Yaskawa INFORM job: small_pipe_cylinder_program.JBI

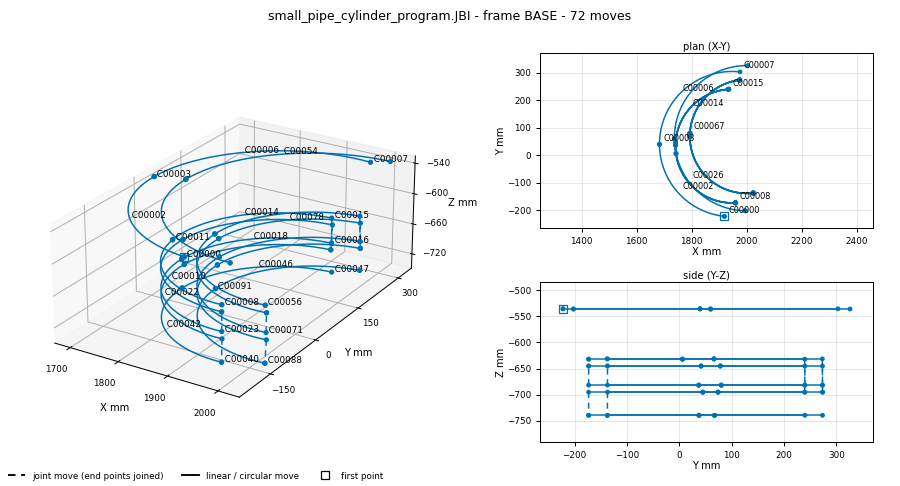
[picture p0: tool path of small_pipe_cylinder_program.JBI in frame BASE, 72 of 105 moves have a stored position in this frame; points joined in program order, loops and branches not executed]
/JOB
//NAME small_pipe_cylinder_program
//POS
///NPOS 96,0,96,0,0,0
///TOOL 0
///POSTYPE BASE
///RECTAN
///RCONF 0,0,0,0,0,0,0,0,0,0,0,0,0,0,0,0,0,0,0,0,0,0,0,0
C00000=1919.180043,-222.253565,-535.692960,175.000000,-60.000000,83.854678
C00001=1919.180043,-222.253565,-535.692960,175.000000,-60.000000,83.854678
C00002=1752.178281,-137.536841,-535.692960,175.000000,-60.000000,42.349745
C00003=1683.223907,39.648654,-535.692960,175.000000,-60.000000,5.000000
C00004=1683.223907,39.648654,-535.692960,175.000000,-60.000000,5.000000
C00005=1683.223907,39.648654,-535.692960,175.000000,-60.000000,5.000000
C00006=1753.745394,220.186963,-535.692960,-175.000000,-60.000000,-42.851744
C00007=1976.266389,303.143966,-535.692960,175.000000,-60.000000,-96.256814
C00008=1960.191811,-173.203258,-631.848500,-86.734427,-89.999999,5.000000
C00009=1960.191811,-173.203258,-631.848500,-86.734427,-89.999999,5.000000
C00010=1829.996385,-136.308422,-631.848500,-124.908956,-89.999999,5.000000
C00011=1743.293664,6.153364,-631.848500,-172.441376,-89.999999,5.000000
C00012=1743.293664,6.153364,-631.848500,-172.441376,-89.999999,5.000000
C00013=1743.293664,6.153364,-631.848500,-172.441376,-89.999999,5.000000
C00014=1789.234673,165.568202,-631.848500,140.288971,-90.000000,5.000000
C00015=1933.789573,239.763101,-631.848500,94.050669,-90.000000,5.000000
C00016=1934.344025,239.801617,-681.511500,93.896764,-90.000000,5.000000
C00017=1934.344025,239.801617,-681.511500,93.896764,-90.000000,5.000000
C00018=1800.374217,177.933006,-681.511500,135.679176,-89.999999,5.000000
C00019=1741.530247,37.146701,-681.511500,175.000000,-89.999999,5.000000
C00020=1741.530247,37.146701,-681.511500,175.000000,-89.999999,5.000000
C00021=1741.530247,37.146701,-681.511500,175.000000,-89.999999,5.000000
C00022=1796.795260,-107.434295,-681.511500,-137.116260,-90.000000,5.000000
C00023=1960.117862,-173.207464,-681.511500,-86.754938,-89.999999,5.000000
C00024=1959.976972,-173.215404,-645.009960,-175.000000,-60.000000,93.205986
C00025=1959.976972,-173.215404,-645.009960,-175.000000,-60.000000,93.205986
C00026=1788.368845,-97.777979,-645.009960,175.000000,-60.000000,39.334277
C00027=1741.661984,41.661903,-645.009960,175.000000,-60.000000,-5.000000
C00028=1741.661984,41.661903,-645.009960,175.000000,-60.000000,-5.000000
C00029=1741.661984,41.661903,-645.009960,175.000000,-60.000000,-5.000000
C00030=1803.493991,181.060147,-645.009960,-175.000000,-60.000000,-45.544034
C00031=1935.364811,239.868614,-645.009960,175.000000,-60.000000,-86.386512
C00032=1933.055266,239.709788,-694.950460,-175.000000,-60.000000,-85.745457
C00033=1933.055266,239.709788,-694.950460,-175.000000,-60.000000,-85.745457
C00034=1804.782266,182.313251,-694.950460,175.000000,-60.000000,-46.041702
C00035=1741.813609,44.834284,-694.950460,175.000000,-60.000000,-5.000000
C00036=1741.813609,44.834284,-694.950460,175.000000,-60.000000,-5.000000
C00037=1741.813609,44.834284,-694.950460,175.000000,-60.000000,-5.000000
C00038=1793.336318,-103.615645,-694.950460,175.000000,-60.000000,41.456964
C00039=1960.430374,-173.189508,-694.950460,175.000000,-60.000000,93.331743
C00040=1959.364741,-173.248787,-739.065960,-175.000000,-60.000000,93.036200
C00041=1959.364741,-173.248787,-739.065960,-175.000000,-60.000000,93.036200
C00042=1802.374489,-113.212580,-739.065960,-175.000000,-60.000000,45.108096
C00043=1741.538277,37.563554,-739.065960,175.000000,-60.000000,-5.000000
C00044=1741.538277,37.563554,-739.065960,175.000000,-60.000000,-5.000000
C00045=1741.538277,37.563554,-739.065960,175.000000,-60.000000,-5.000000
C00046=1807.515538,184.901335,-739.065960,-175.000000,-60.000000,-47.084060
C00047=1935.638086,239.885690,-739.065960,175.000000,-60.000000,-86.462333
C00048=1995.134330,-202.194927,-536.078460,175.000000,-60.000000,88.606450
C00049=1995.134330,-202.194927,-536.078460,175.000000,-60.000000,88.606450
C00050=1813.082954,-123.234912,-536.078460,175.000000,-60.000000,44.498499
C00051=1737.325476,59.695630,-536.078460,-175.000000,-60.000000,5.000000
C00052=1737.325476,59.695630,-536.078460,-175.000000,-60.000000,5.000000
C00053=1737.325476,59.695630,-536.078460,-175.000000,-60.000000,5.000000
C00054=1817.601589,251.667664,-536.078460,-175.000000,-60.000000,-45.879584
C00055=2004.328239,326.202425,-536.078460,-175.000000,-60.000000,-90.600098
C00056=2023.008270,-137.447122,-631.340500,-83.760239,-90.000000,5.000000
C00057=2023.008270,-137.447122,-631.340500,-83.760239,-90.000000,5.000000
C00058=1844.451298,-67.609986,-631.340500,-138.962647,-89.999999,5.000000
C00059=1793.619781,66.206992,-631.340500,-175.000000,-89.999999,5.000000
C00060=1793.619781,66.206992,-631.340500,-175.000000,-89.999999,5.000000
C00061=1793.619781,66.206992,-631.340500,-175.000000,-89.999999,5.000000
C00062=1827.332269,181.452385,-631.340500,146.826604,-89.999999,5.000000
C00063=1973.123011,273.324532,-631.340500,97.608744,-89.999999,5.000000
C00064=1974.788266,273.540110,-681.475500,97.143765,-90.000000,5.000000
C00065=1974.788266,273.540110,-681.475500,97.143765,-90.000000,5.000000
C00066=1849.340238,209.503950,-681.475500,136.941193,-90.000000,5.000000
C00067=1793.957901,80.233327,-681.475500,175.000000,-90.000000,5.000000
C00068=1793.957901,80.233327,-681.475500,175.000000,-90.000000,5.000000
C00069=1793.957901,80.233327,-681.475500,175.000000,-90.000000,5.000000
C00070=1870.223695,-92.494769,-681.475500,-129.029688,-90.000000,5.000000
C00071=2024.730486,-137.251517,-681.475500,-83.280269,-90.000000,5.000000
C00072=2025.322950,-137.180845,-644.921960,175.000000,-60.000000,96.884954
C00073=2025.322950,-137.180845,-644.921960,175.000000,-60.000000,96.884954
C00074=1848.138782,-71.733732,-644.921960,175.000000,-60.000000,42.569271
C00075=1793.863419,78.477670,-644.921960,-175.000000,-60.000000,-5.000000
C00076=1793.863419,78.477670,-644.921960,-175.000000,-60.000000,-5.000000
C00077=1793.863419,78.477670,-644.921960,-175.000000,-60.000000,-5.000000
C00078=1854.789412,215.118781,-644.921960,-175.000000,-60.000000,-45.225583
C00079=1974.546352,273.509645,-644.921960,-175.000000,-60.000000,-82.788717
C00080=1975.515287,273.629922,-694.925960,-175.000000,-60.000000,-83.059086
C00081=1975.515287,273.629922,-694.925960,-175.000000,-60.000000,-83.059086
C00082=1852.242914,212.547679,-694.925960,175.000000,-60.000000,-44.223499
C00083=1793.692664,74.091023,-694.925960,175.000000,-60.000000,-5.000000
C00084=1793.692664,74.091023,-694.925960,175.000000,-60.000000,-5.000000
C00085=1793.692664,74.091023,-694.925960,175.000000,-60.000000,-5.000000
C00086=1859.683120,-83.344030,-694.925960,175.000000,-60.000000,47.104301
C00087=2025.338332,-137.178987,-694.925960,-175.000000,-60.000000,96.889245
C00088=2022.883642,-137.460710,-739.166460,175.000000,-60.000000,96.205045
C00089=2022.883642,-137.460710,-739.166460,175.000000,-60.000000,96.205045
C00090=1857.753393,-81.527923,-739.166460,175.000000,-60.000000,46.370500
C00091=1793.612010,67.285889,-739.166460,175.000000,-60.000000,5.000000
C00092=1793.612010,67.285889,-739.166460,175.000000,-60.000000,5.000000
C00093=1793.612010,67.285889,-739.166460,175.000000,-60.000000,5.000000
C00094=1851.248443,211.518786,-739.166460,175.000000,-60.000000,-43.827253
C00095=1975.230312,273.595029,-739.166460,175.000000,-60.000000,-82.979584
///POSTYPE PULSE
///PULSE
EX00000=86016.0
EX00001=95232.0
EX00002=275456.0
EX00003=283648.0
///POSTYPE PULSE
///PULSE
EC00000=86016.0
EC00001=86016.0
EC00002=86016.0
EC00003=86016.0
EC00004=86016.0
EC00005=86016.0
EC00006=86016.0
EC00007=86016.0
EC00008=95232.0
EC00009=95232.0
EC00010=95232.0
EC00011=95232.0
EC00012=95232.0
EC00013=95232.0
EC00014=95232.0
EC00015=95232.0
EC00016=95232.0
EC00017=95232.0
EC00018=95232.0
EC00019=95232.0
EC00020=95232.0
EC00021=95232.0
EC00022=95232.0
EC00023=95232.0
EC00024=95232.0
EC00025=95232.0
EC00026=95232.0
EC00027=95232.0
EC00028=95232.0
EC00029=95232.0
EC00030=95232.0
EC00031=95232.0
EC00032=95232.0
EC00033=95232.0
EC00034=95232.0
EC00035=95232.0
EC00036=95232.0
EC00037=95232.0
EC00038=95232.0
EC00039=95232.0
EC00040=95232.0
EC00041=95232.0
EC00042=95232.0
EC00043=95232.0
EC00044=95232.0
EC00045=95232.0
EC00046=95232.0
EC00047=95232.0
EC00048=275456.0
EC00049=275456.0
EC00050=275456.0
EC00051=275456.0
EC00052=275456.0
EC00053=275456.0
EC00054=275456.0
EC00055=275456.0
EC00056=283648.0
EC00057=283648.0
EC00058=283648.0
EC00059=283648.0
EC00060=283648.0
EC00061=283648.0
EC00062=283648.0
EC00063=283648.0
EC00064=283648.0
EC00065=283648.0
EC00066=283648.0
EC00067=283648.0
EC00068=283648.0
EC00069=283648.0
EC00070=283648.0
EC00071=283648.0
EC00072=283648.0
EC00073=283648.0
EC00074=283648.0
EC00075=283648.0
EC00076=283648.0
EC00077=283648.0
EC00078=283648.0
EC00079=283648.0
EC00080=283648.0
EC00081=283648.0
EC00082=283648.0
EC00083=283648.0
EC00084=283648.0
EC00085=283648.0
EC00086=283648.0
EC00087=283648.0
EC00088=283648.0
EC00089=283648.0
EC00090=283648.0
EC00091=283648.0
EC00092=283648.0
EC00093=283648.0
EC00094=283648.0
EC00095=283648.0
//INST
///DATE 2023/08/16 14:27
///ATTR SC,RW,RJ
////FRAME BASE
///GROUP1 RB1,ST1
NOP
MOVJ P009 EX000 VJ=15.00
MOVJ C00000 EC00000 VJ=15.0
CALL JOB:SPYON
MOVC C00001 EC00001 V=150.0
MOVC C00002 EC00002 V=150.0
MOVC C00003 EC00003 V=150.0
MOVJ C00004 EC00004 VJ=15.0
MOVC C00005 EC00005 V=150.0
MOVC C00006 EC00006 V=150.0
MOVC C00007 EC00007 V=150.0
CALL JOB:SPYOF
MOVJ P009 VJ=15.00
MOVL P009 EX00000 V=150.0
MOVJ C00008 EC00008 VJ=15.0
CALL JOB:SPYON
MOVC C00009 EC00009 V=150.0
MOVC C00010 EC00010 V=150.0
MOVC C00011 EC00011 V=150.0
MOVJ C00012 EC00012 VJ=15.0
MOVC C00013 EC00013 V=150.0
MOVC C00014 EC00014 V=150.0
MOVC C00015 EC00015 V=150.0
MOVJ C00016 EC00016 VJ=15.0
MOVC C00017 EC00017 V=150.0
MOVC C00018 EC00018 V=150.0
MOVC C00019 EC00019 V=150.0
MOVJ C00020 EC00020 VJ=15.0
MOVC C00021 EC00021 V=150.0
MOVC C00022 EC00022 V=150.0
MOVC C00023 EC00023 V=150.0
MOVJ C00024 EC00024 VJ=15.0
MOVC C00025 EC00025 V=150.0
MOVC C00026 EC00026 V=150.0
MOVC C00027 EC00027 V=150.0
MOVJ C00028 EC00028 VJ=15.0
MOVC C00029 EC00029 V=150.0
MOVC C00030 EC00030 V=150.0
MOVC C00031 EC00031 V=150.0
MOVJ C00032 EC00032 VJ=15.0
MOVC C00033 EC00033 V=150.0
MOVC C00034 EC00034 V=150.0
MOVC C00035 EC00035 V=150.0
MOVJ C00036 EC00036 VJ=15.0
MOVC C00037 EC00037 V=150.0
MOVC C00038 EC00038 V=150.0
MOVC C00039 EC00039 V=150.0
MOVJ C00040 EC00040 VJ=15.0
MOVC C00041 EC00041 V=150.0
MOVC C00042 EC00042 V=150.0
MOVC C00043 EC00043 V=150.0
MOVJ C00044 EC00044 VJ=15.0
MOVC C00045 EC00045 V=150.0
MOVC C00046 EC00046 V=150.0
MOVC C00047 EC00047 V=150.0
CALL JOB:SPYOF
MOVJ P009 VJ=15.00
MOVL P009 EX00001 V=150.0
MOVJ C00048 EC00048 VJ=15.0
CALL JOB:SPYON
MOVC C00049 EC00049 V=150.0
MOVC C00050 EC00050 V=150.0
MOVC C00051 EC00051 V=150.0
MOVJ C00052 EC00052 VJ=15.0
MOVC C00053 EC00053 V=150.0
MOVC C00054 EC00054 V=150.0
MOVC C00055 EC00055 V=150.0
CALL JOB:SPYOF
MOVJ P009 VJ=15.00
MOVL P009 EX00002 V=150.0
MOVJ C00056 EC00056 VJ=15.0
CALL JOB:SPYON
MOVC C00057 EC00057 V=150.0
MOVC C00058 EC00058 V=150.0
MOVC C00059 EC00059 V=150.0
MOVJ C00060 EC00060 VJ=15.0
MOVC C00061 EC00061 V=150.0
MOVC C00062 EC00062 V=150.0
MOVC C00063 EC00063 V=150.0
MOVJ C00064 EC00064 VJ=15.0
MOVC C00065 EC00065 V=150.0
MOVC C00066 EC00066 V=150.0
MOVC C00067 EC00067 V=150.0
MOVJ C00068 EC00068 VJ=15.0
MOVC C00069 EC00069 V=150.0
MOVC C00070 EC00070 V=150.0
MOVC C00071 EC00071 V=150.0
MOVJ C00072 EC00072 VJ=15.0
MOVC C00073 EC00073 V=150.0
MOVC C00074 EC00074 V=150.0
MOVC C00075 EC00075 V=150.0
MOVJ C00076 EC00076 VJ=15.0
MOVC C00077 EC00077 V=150.0
MOVC C00078 EC00078 V=150.0
MOVC C00079 EC00079 V=150.0
MOVJ C00080 EC00080 VJ=15.0
MOVC C00081 EC00081 V=150.0
MOVC C00082 EC00082 V=150.0
MOVC C00083 EC00083 V=150.0
MOVJ C00084 EC00084 VJ=15.0
MOVC C00085 EC00085 V=150.0
MOVC C00086 EC00086 V=150.0
MOVC C00087 EC00087 V=150.0
MOVJ C00088 EC00088 VJ=15.0
MOVC C00089 EC00089 V=150.0
MOVC C00090 EC00090 V=150.0
MOVC C00091 EC00091 V=150.0
MOVJ C00092 EC00092 VJ=15.0
MOVC C00093 EC00093 V=150.0
MOVC C00094 EC00094 V=150.0
MOVC C00095 EC00095 V=150.0
CALL JOB:SPYOF
MOVJ P009 VJ=15.00
MOVL P009 EX00003 V=150.0
END
